// TIA Portal V18 export
TYPE "UDT_HCsAI"
// stored: IsFailsafeCompliant false
   STRUCT
      rSupplyWaterTemp : Array[1..2] of Real;
      rReturnWaterTemp : Array[1..2] of Real;
      r3vwPosFbk : Array[1..2] of Real;
   END_STRUCT;
END_TYPE
